RESOURCE RES0 : EMB_RES_ECO
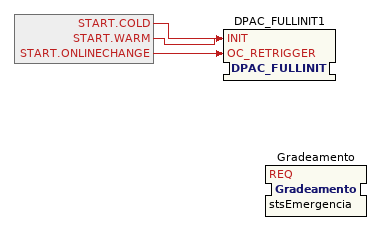
  FBS
    Gradeamento : Gradeamento;
    DPAC_FULLINIT1 : DPAC_FULLINIT;
  END_FBS
  EVENT_CONNECTIONS
    START.COLD TO DPAC_FULLINIT1.INIT;
    START.WARM TO DPAC_FULLINIT1.INIT;
    START.ONLINECHANGE TO DPAC_FULLINIT1.OC_RETRIGGER;
  END_CONNECTIONS
END_RESOURCE
